ABB RAPID module: wObj_AreaBuffers1.mod

MODULE wObj_AreaBuffers1
	! Points are read in order of declaration.
  ! Please do not change the order of points!

  LOCAL PERS robtarget pWobj_U_PointX1:=[[1984.387,-1236.534,81.74384],[0.0242001302540302,-0.101351700723171,0.994550466537476,0.00339692528359592],[-1,0,-1,0],[9E+09,9E+09,9E+09,9E+09,9E+09,9E+09]];
	LOCAL PERS robtarget pWobj_U_PointX2:=[[-1649.67,-1018.287,81.20656],[0.0209988243877888,0.545415043830872,0.837809264659882,-0.0125325759872794],[-2,0,-1,0],[9E+09,9E+09,9E+09,9E+09,9E+09,9E+09]];
	LOCAL PERS robtarget pWobj_U_PointY1:=[[1921.615,-2197.818,94.29008],[0.00870867632329464,0.514756858348846,0.856986582279205,0.022882092744112],[-1,0,0,0],[9E+09,9E+09,9E+09,9E+09,9E+09,9E+09]];

ENDMODULE
